// TIA Portal V20 export
TYPE "UDT_control"
   STRUCT
      resetCounters { ExternalVisible := 'False'} : DInt;   // 1: cmd active
      startTaktTimeCnt { ExternalVisible := 'False'} : DInt;   // 1: cmd active
      stopTaktTimeCnt { ExternalVisible := 'False'} : DInt;   // 1: cmd active
      actualMinus1 : DInt;
      actualPlus1 : DInt;
   END_STRUCT;
END_TYPE
